// TIA Portal project "SMTest" (V16)

(* hardware
DEVICE "S7-1200 station_1"  S7-1200 Station
   slot 0: "Rack_0"  S7-1200 Rack  Rack  V1.0
   slot 1: "PLC_1"  CPU 1212C AC/DC/Rly  6ES7 212-1BE40-0XB0  V4.4
*)

// ===== PLC "PLC_1"  CPU 1212C AC/DC/Rly =====

VAR_GLOBAL   // PLC tag table "Default tag table"
   "System_Byte" AT %MB1 : Byte;
   "FirstScan" AT %M1.0 : Bool;
   "DiagStatusUpdate" AT %M1.1 : Bool;
   "AlwaysTRUE" AT %M1.2 : Bool;
   "AlwaysFALSE" AT %M1.3 : Bool;
END_VAR

VAR_GLOBAL   // PLC tag table "State"
   "State 0" AT %M2.0 : Bool;
   "State 1" AT %M2.1 : Bool;
   "State 2" AT %M2.2 : Bool;
   "State 3" AT %M2.3 : Bool;
   "State 4" AT %M2.4 : Bool;
   "State 5" AT %M2.5 : Bool;
   "State 6" AT %M2.6 : Bool;
   "State 7" AT %M2.7 : Bool;
   "SS" AT %MB0 : Byte;   // SAVED STATE
END_VAR

VAR_GLOBAL   // PLC tag table "Buttons"
   "Start" AT %I0.0 : Bool;
   "Stop" AT %I0.4 : Bool;
   "Drain" AT %I0.5 : Bool;
   "Emergency" AT %I0.6 : Bool;
END_VAR

VAR_GLOBAL   // PLC tag table "Sensors"
   "WL1" AT %I0.1 : Bool;   // WATER LEVEL LOW
   "WL2" AT %I0.2 : Bool;   // WATER LEVEL HIGH
   "CH1" AT %I0.3 : Bool;   // CHLORINE LEVEL
END_VAR

VAR_GLOBAL   // PLC tag table "Actuators"
   "PM1" AT %Q0.4 : Bool;   // Pump Water Intake
   "PM2" AT %Q0.5 : Bool;   // Pump Water Drain
   "PM3" AT %Q0.6 : Bool;   // Pump Emergency Drain
   "PM4" AT %Q0.7 : Bool;   // Pump Chrorine Supply
   "M1" AT %Q1.0 : Bool;   // Mixer Motor
END_VAR

VAR_GLOBAL   // PLC tag table "Indicators"
   "HL1" AT %Q0.0 : Bool;   // LAMP WORK
   "HL2" AT %Q0.1 : Bool;   // LAMP STOP
   "HL3" AT %Q0.2 : Bool;   // LAMP EMERGENCY STOP
   "HL4" AT %Q0.3 : Bool;   // EMERGENCY DRAIN
END_VAR

// folder: System blocks/Program resources

DATA_BLOCK "Purification"   // DB1
{ S7_Optimized_Access := 'TRUE' }
AUTHOR : Simatic
FAMILY : IEC
NAME : IEC_TMR
VERSION : 1.0
// stored: InstanceOfName IEC_TIMER
"IEC_TIMER"
BEGIN
END_DATA_BLOCK

// folder: (top level)

ORGANIZATION_BLOCK "Main"   // OB1, LAD, ProgramCycle
TITLE = "Main Program Sweep (Cycle)"
{ S7_Optimized_Access := 'TRUE' }
VERSION : 0.1
   VAR_INPUT
      Initial_Call : Bool;   // Initial call of this OB
      Remanence : Bool;   // =True, if remanent data are available
   END_VAR
   VAR_TEMP   // added for the SCL form of the ladder/FBD networks
      _w1 : Bool;
      _w2 : Bool;
      _w3 : Bool;
      _w4 : Bool;
      _w5 : Bool;
      _w6 : Bool;
      _w7 : Bool;
      _w8 : Bool;
      _w9 : Bool;
   END_VAR
BEGIN

REGION Network 1: Initialization
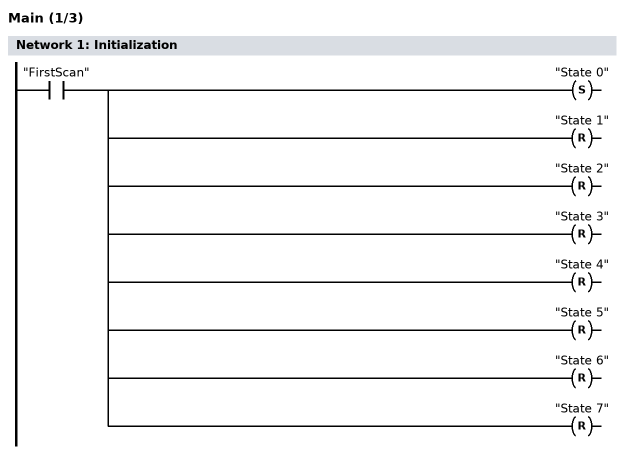
   RUNG wire#powerrail
      Contact( "FirstScan" )
      wire#w1
      S_Coil( "State 0" )
   END_RUNG
   RUNG wire#w1
      R_Coil( "State 1" )
   END_RUNG
   RUNG wire#w1
      R_Coil( "State 2" )
   END_RUNG
   RUNG wire#w1
      R_Coil( "State 3" )
   END_RUNG
   RUNG wire#w1
      R_Coil( "State 4" )
   END_RUNG
   RUNG wire#w1
      R_Coil( "State 5" )
   END_RUNG
   RUNG wire#w1
      R_Coil( "State 6" )
   END_RUNG
   RUNG wire#w1
      R_Coil( "State 7" )
   END_RUNG
   // the same network as SCL:
   IF "FirstScan" THEN
       "State 0" := TRUE;
       "State 1" := FALSE;
       "State 2" := FALSE;
       "State 3" := FALSE;
       "State 4" := FALSE;
       "State 5" := FALSE;
       "State 6" := FALSE;
       "State 7" := FALSE;
   END_IF;
END_REGION

REGION Network 2: State Machine
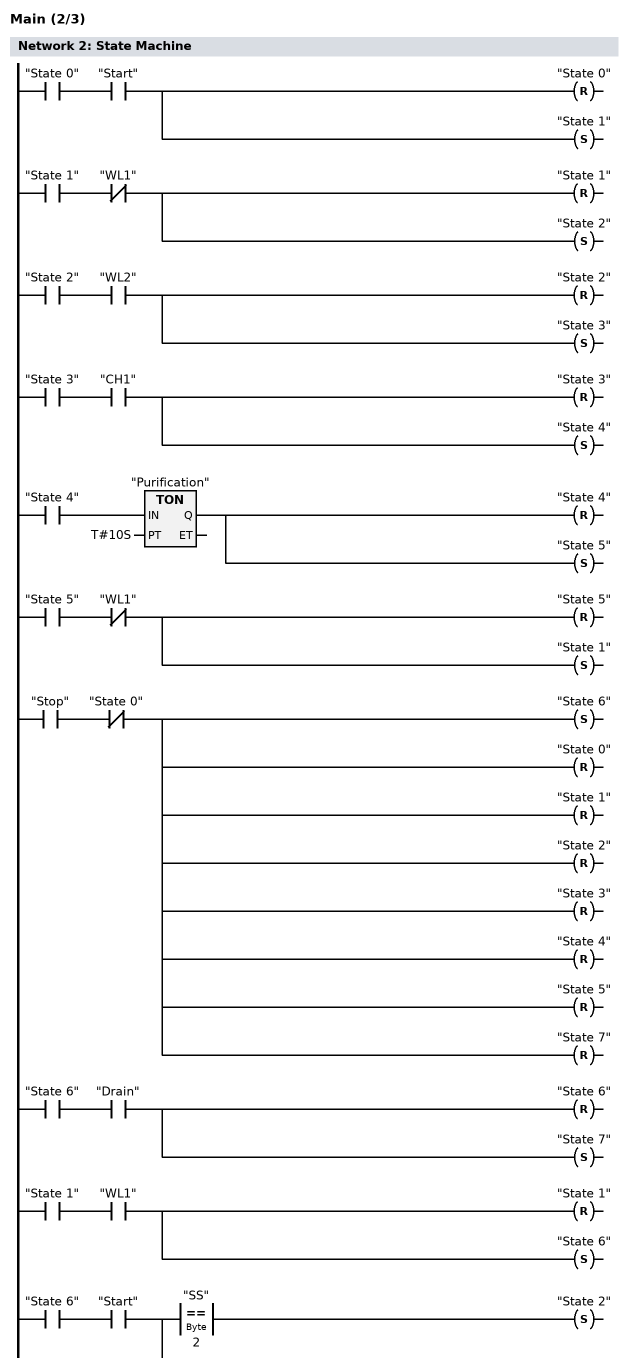
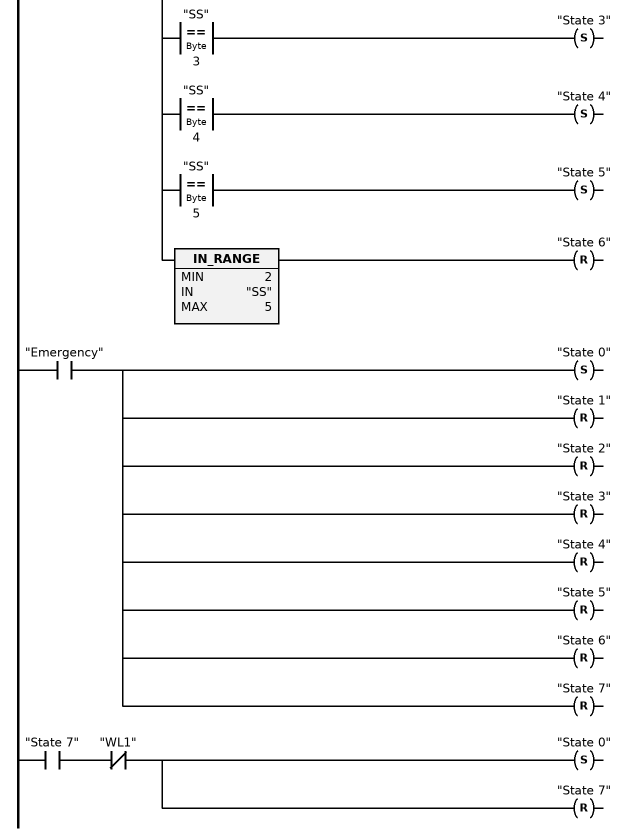
   #_w1 := "State 0" AND "Start";
   IF #_w1 THEN
       "State 0" := FALSE;
       "State 1" := TRUE;
   END_IF;
   #_w2 := "State 1" AND NOT "WL1";
   IF #_w2 THEN
       "State 1" := FALSE;
       "State 2" := TRUE;
   END_IF;
   #_w3 := "State 2" AND "WL2";
   IF #_w3 THEN
       "State 2" := FALSE;
       "State 3" := TRUE;
   END_IF;
   #_w4 := "State 3" AND "CH1";
   IF #_w4 THEN
       "State 3" := FALSE;
       "State 4" := TRUE;
   END_IF;
   "Purification".TON(IN := "State 4", PT := T#10S);
   IF "Purification".Q THEN
       "State 4" := FALSE;
       "State 5" := TRUE;
   END_IF;
   #_w5 := "State 5" AND NOT "WL1";
   IF #_w5 THEN
       "State 5" := FALSE;
       "State 1" := TRUE;
   END_IF;
   IF "Stop" AND NOT "State 0" THEN "State 6" := TRUE; END_IF;
   #_w6 := "Stop" AND NOT "State 0";
   IF #_w6 THEN
       "State 0" := FALSE;
       "State 1" := FALSE;
       "State 2" := FALSE;
       "State 3" := FALSE;
       "State 4" := FALSE;
       "State 5" := FALSE;
       "State 7" := FALSE;
   END_IF;
   #_w7 := "State 6" AND "Drain";
   IF #_w7 THEN
       "State 6" := FALSE;
       "State 7" := TRUE;
   END_IF;
   #_w8 := "State 1" AND "WL1";
   IF #_w8 THEN
       "State 1" := FALSE;
       "State 6" := TRUE;
   END_IF;
   #_w9 := "State 6" AND "Start";
   IF #_w9 AND ("SS" = 2) THEN "State 2" := TRUE; END_IF;
   IF #_w9 AND ("SS" = 3) THEN "State 3" := TRUE; END_IF;
   IF #_w9 AND ("SS" = 4) THEN "State 4" := TRUE; END_IF;
   IF #_w9 AND ("SS" = 5) THEN "State 5" := TRUE; END_IF;
   IF #_w9 AND (2 <= "SS") AND ("SS" <= 5) THEN "State 6" := FALSE; END_IF;
   IF "Emergency" THEN
       "State 0" := TRUE;
       "State 1" := FALSE;
       "State 2" := FALSE;
       "State 3" := FALSE;
       "State 4" := FALSE;
       "State 5" := FALSE;
       "State 6" := FALSE;
       "State 7" := FALSE;
   END_IF;
   IF "State 7" AND NOT "WL1" THEN
       "State 0" := TRUE;
       "State 7" := FALSE;
   END_IF;
END_REGION

REGION Network 3: Busines Logic
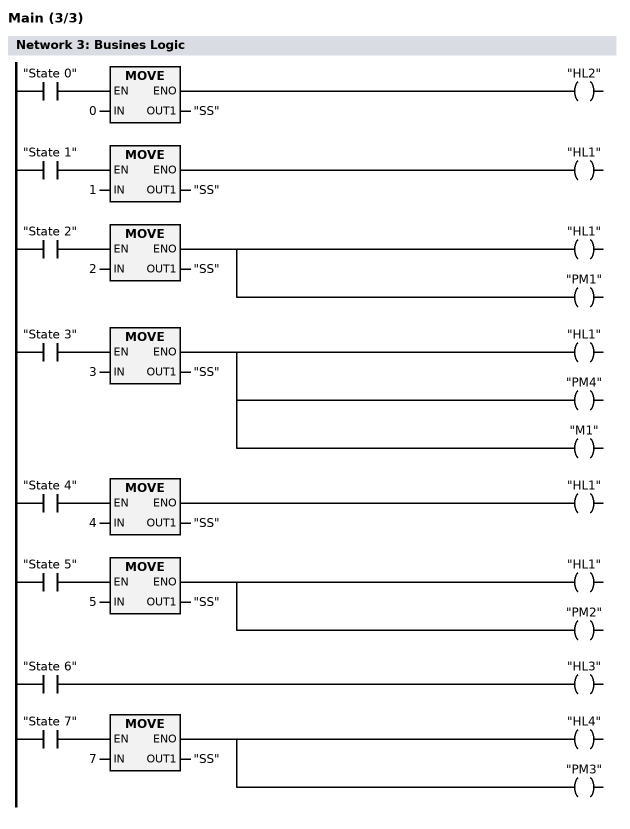
   RUNG wire#powerrail
      Contact( "State 0" )
      Move(in := 0, out1 => "SS")
      Coil( "HL2" )
   END_RUNG
   RUNG wire#powerrail
      Contact( "State 1" )
      Move(in := 1, out1 => "SS")
      Coil( "HL1" )
   END_RUNG
   RUNG wire#powerrail
      Contact( "State 2" )
      Move(in := 2, out1 => "SS")
      wire#w1
      Coil( "HL1" )
   END_RUNG
   RUNG wire#w1
      Coil( "PM1" )
   END_RUNG
   RUNG wire#powerrail
      Contact( "State 3" )
      Move(in := 3, out1 => "SS")
      wire#w2
      Coil( "HL1" )
   END_RUNG
   RUNG wire#w2
      Coil( "PM4" )
   END_RUNG
   RUNG wire#w2
      Coil( "M1" )
   END_RUNG
   RUNG wire#powerrail
      Contact( "State 4" )
      Move(in := 4, out1 => "SS")
      Coil( "HL1" )
   END_RUNG
   RUNG wire#powerrail
      Contact( "State 5" )
      Move(in := 5, out1 => "SS")
      wire#w3
      Coil( "HL1" )
   END_RUNG
   RUNG wire#w3
      Coil( "PM2" )
   END_RUNG
   RUNG wire#powerrail
      Contact( "State 6" )
      Coil( "HL3" )
   END_RUNG
   RUNG wire#powerrail
      Contact( "State 7" )
      Move(in := 7, out1 => "SS")
      wire#w4
      Coil( "HL4" )
   END_RUNG
   RUNG wire#w4
      Coil( "PM3" )
   END_RUNG
   // the same network as SCL:
   IF "State 0" THEN "SS" := 0; END_IF;
   "HL2" := "State 0";
   IF "State 1" THEN "SS" := 1; END_IF;
   "HL1" := "State 1";
   IF "State 2" THEN "SS" := 2; END_IF;
   "HL1" := "State 2";
   "PM1" := "State 2";
   IF "State 3" THEN "SS" := 3; END_IF;
   "HL1" := "State 3";
   "PM4" := "State 3";
   "M1" := "State 3";
   IF "State 4" THEN "SS" := 4; END_IF;
   "HL1" := "State 4";
   IF "State 5" THEN "SS" := 5; END_IF;
   "HL1" := "State 5";
   "PM2" := "State 5";
   "HL3" := "State 6";
   IF "State 7" THEN "SS" := 7; END_IF;
   "HL4" := "State 7";
   "PM3" := "State 7";
END_REGION
END_ORGANIZATION_BLOCK